FUNCTION StateTop : BOOL
VAR_INPUT
END_VAR
VAR
END_VAR

END_FUNCTION

(* stored: Version 1.1.0.1, ProductVersion 3.1.4022.18
   POU StateTop: Id {47de2e36-77f3-40e1-8166-734388e1c343}, SpecialFunc None *)
